(* IEC 61131-3 sources: plc_generation_empirical_study/datasets/task_bank_lean_runtime_v0_1/tasks/C04_R21_lean_composite, 2 files *)

(* ---- interface.st ---- *)
FUNCTION_BLOCK C04_R21_lean_composite
VAR_INPUT
    A_EventA : BOOL;
    A_EventB : BOOL;
    A_Qualify : BOOL;
    A_Inhibit : BOOL;
    A_Reset : BOOL;
    A_MaxCount : INT;
    B_Info : BOOL;
    B_Warning : BOOL;
    B_Trip : BOOL;
    B_Emergency : BOOL;
    B_Suppress : BOOL;
    SubsystemBEnable : BOOL;
    CrossReset : BOOL;
END_VAR
VAR_OUTPUT
    A_PulseA : BOOL;
    A_PulseB : BOOL;
    A_Count : INT;
    A_Locked : BOOL;
    A_LastSource : INT;
    B_Active : BOOL;
    B_Level : INT;
    CrossReady : BOOL;
    CrossBlocked : BOOL;
END_VAR
END_FUNCTION_BLOCK

(* ---- reference.st ---- *)
FUNCTION_BLOCK C04_R21_lean_composite
VAR_INPUT
    A_EventA : BOOL;
    A_EventB : BOOL;
    A_Qualify : BOOL;
    A_Inhibit : BOOL;
    A_Reset : BOOL;
    A_MaxCount : INT;
    B_Info : BOOL;
    B_Warning : BOOL;
    B_Trip : BOOL;
    B_Emergency : BOOL;
    B_Suppress : BOOL;
    SubsystemBEnable : BOOL;
    CrossReset : BOOL;
END_VAR
VAR_OUTPUT
    A_PulseA : BOOL;
    A_PulseB : BOOL;
    A_Count : INT;
    A_Locked : BOOL;
    A_LastSource : INT;
    B_Active : BOOL;
    B_Level : INT;
    CrossReady : BOOL;
    CrossBlocked : BOOL;
END_VAR
VAR
    A_PrevA : BOOL;
    A_PrevB : BOOL;
END_VAR

A_PulseA := FALSE;
A_PulseB := FALSE;
IF A_Reset AND (NOT A_EventA) AND (NOT A_EventB) THEN
    A_Count := 0;
    A_Locked := FALSE;
    A_LastSource := 0;
ELSIF A_MaxCount <= 0 THEN
    A_Locked := TRUE;
ELSIF A_Qualify AND (NOT A_Inhibit) AND (NOT A_Locked) THEN
    IF A_EventA AND (NOT A_PrevA) THEN
        A_PulseA := TRUE;
        A_Count := A_Count + 1;
        A_LastSource := 1;
    ELSIF A_EventB AND (NOT A_PrevB) THEN
        A_PulseB := TRUE;
        A_Count := A_Count + 1;
        A_LastSource := 2;
    END_IF;
    IF A_Count >= A_MaxCount THEN A_Count := A_MaxCount; A_Locked := TRUE; END_IF;
END_IF;
A_PrevA := A_EventA;
A_PrevB := A_EventB;

IF CrossReset THEN
    CrossReady := FALSE;
ELSIF A_PulseA THEN
    CrossReady := TRUE;
END_IF;
CrossBlocked := SubsystemBEnable AND (NOT CrossReady);

IF SubsystemBEnable AND CrossReady THEN
    IF B_Emergency THEN
        B_Level := 4;
        B_Active := TRUE;
    ELSIF B_Suppress THEN
        B_Level := 0;
        B_Active := FALSE;
    ELSIF B_Trip THEN
        B_Level := 3;
        B_Active := TRUE;
    ELSIF B_Warning THEN
        B_Level := 2;
        B_Active := TRUE;
    ELSIF B_Info THEN
        B_Level := 1;
        B_Active := TRUE;
    ELSE
        B_Level := 0;
        B_Active := FALSE;
    END_IF;
ELSE
    B_Active := FALSE;
    B_Level := 0;
END_IF;

END_FUNCTION_BLOCK
